{region '#Template'}
	{attribute 'Version' := '5.0.1.0'}
	{attribute 'Tags' := '"LCID": "1031", "Text": "AC, Aggregates, Cooler, Temperature"'}
	{attribute 'Tags' := '"LCID": "1033", "Text": "AC, Aggregates, Cooler, Temperature"'}
	{attribute 'Description' := '"LCID": "1031", "Text": "Aggregat Kühler Temperatur mit Ventil"'}
	{attribute 'Description' := '"LCID": "1033", "Text": "Aggregate cooler temperature with valve"'}
{endregion}
FUNCTION_BLOCK FB_BA_AC_ColT_02 EXTENDS FB_BA_View
VAR_INPUT
	fSpTSuA					: REAL;// Sollwert Temperatur kühlen // Setpoint temperature cooling
	fTSuA					: REAL;// Zuluft Temperatur // Supply air temperature
	bSyncTSuACtrl			: BOOL;
	fSyncTSuACtrl			: REAL;		
	stCmd					: ST_BA_Binary;				
END_VAR
VAR_OUTPUT
	fPresentValue			: REAL;	
	bActiveSeqCtrl			: BOOL;
END_VAR
VAR_IN_OUT
	stTSeqLink			: ST_BA_SeqLink;	//	Sequenz Link Struktur	//	Sequence link structure	
END_VAR
VAR_INPUT CONSTANT PERSISTENT
END_VAR
VAR_INPUT CONSTANT
	TFl						: FB_BA_SensorAnalog;												
	TRt						: FB_BA_SensorAnalog;			
	TSuACtrl				: FB_BA_AC_ColTSuACtrl;
	Vlv						: FB_BA_Vlv;
	PlantLock				: FB_BA_PlantLock;																							
END_VAR
VAR		
	bPrioSfty				: BOOL;
	bPrioCrit				: BOOL;		
	PrioSwiVal				: FB_BA_PrioSwi_B04;	
END_VAR
VAR // added by the converter: edge detectors and wires of the graphical bodies
    _s1 : ST_BA_Analog;
END_VAR

SUPER^(); // FB_BA_View
PlantLock(); // FB_BA_PlantLock
bPrioSfty := PlantLock.bPrioHigh OR PlantLock.bPrioLocalHigh;
bPrioCrit := PlantLock.bPrioMedium OR PlantLock.bPrioLocalMedium;
TFl(); // FB_BA_SensorAnalog
TRt(); // FB_BA_SensorAnalog
PrioSwiVal(
    bEn01 := stCmd.bEnSfty,
    bVal01 := stCmd.bValSfty,
    bEn02 := stCmd.bEnCrit,
    bVal02 := stCmd.bValCrit,
    bEn03 := stCmd.bEnPgm,
    bVal03 := stCmd.bValPgm); // FB_BA_PrioSwi_B04
TSuACtrl(
    bEn := PrioSwiVal.bVal,
    fSpTSuA := fSpTSuA,
    fTSuA := fTSuA,
    bSync := bSyncTSuACtrl,
    fSync := fSyncTSuACtrl,
    stSeqLink := stTSeqLink); // FB_BA_AC_ColTSuACtrl
bActiveSeqCtrl := TSuACtrl.bIsActive;
// compose _s1 : ST_BA_Analog
_s1.bEnSfty := stCmd.bEnSfty OR bPrioSfty;
_s1.fValSfty := TSuACtrl.fY;
_s1.bEnCrit := stCmd.bEnCrit OR bPrioCrit;
_s1.fValCrit := TSuACtrl.fY;
_s1.bEnPgm := stCmd.bEnPgm;
_s1.fValPgm := TSuACtrl.fY;
Vlv(stCmd := _s1); // FB_BA_Vlv
fPresentValue := Vlv.fMdlt;

METHOD FB_init : BOOL
VAR_INPUT
	bInitRetains : BOOL; // if TRUE, the retain variables are initialized (warm start / cold start)
	bInCopyCode : BOOL;  // if TRUE, the instance afterwards gets moved into the copy code (online change)
END_VAR
PlantLock.Parent								:= THIS^;		

TFl.iParent								:= THIS^;		
TFl.iLabel								:= LblAgg_TemperatureFlow;   
TFl.sObjectName							:= '{Idx=41}';						 
TFl.eDPADMode							:= E_BA_DPADMode.eInclude;															
TFl.MV.eUnit							:= E_BA_Unit.eTemperature_DegreesCelsius;
TFl.MV.fResolution 						:= 0.01;
TFl.MV.fScaleOffset 					:= 0; 
TFl.MV.bEventDetectionEnable			:= TRUE;
TFl.MV.eEnPlantLock						:= E_BA_LockPriority.eNoLock;

TRt.iParent								:= THIS^;		
TRt.iLabel								:= LblAgg_TemperatureReturnFlow;
TRt.sObjectName							:= '{Idx=41}';						 
TRt.eDPADMode							:= E_BA_DPADMode.eInclude;																												
TRt.MV.eUnit							:= E_BA_Unit.eTemperature_DegreesCelsius;
TRt.MV.fResolution 						:= 0.01;
TRt.MV.fScaleOffset 					:= 0;  
TRt.MV.bEventDetectionEnable			:= TRUE;	
TRt.MV.eEnPlantLock						:= E_BA_LockPriority.eNoLock;

TSuACtrl.iParent						:= THIS^;	 
TSuACtrl.iLabel							:= LblCtl_SupplyAirTemperatureControl;
TSuACtrl.sObjectName					:= '{Idx=41}';						 
TSuACtrl.eDPADMode						:= E_BA_DPADMode.eInclude;								
                        				
Vlv.iParent								:= THIS^;
Vlv.iLabel								:= LblAgg_Valve;
Vlv.sObjectName							:= '{Idx=41}';						 
Vlv.eDPADMode							:= E_BA_DPADMode.eInclude;
END_METHOD

END_FUNCTION_BLOCK

(* stored: Version 1.1.0.1, ProductVersion 3.1.4024.12
   POU FB_BA_AC_ColT_02: Id {866681a9-ff68-4603-9647-0c1b945954cb}, SpecialFunc None
   Method FB_init: Id {b64f6103-0d34-457a-bb3c-2b6bc3ad8ec8} *)
